// TIA Portal V16 program export: 1 tag tables, 0 data types, 0 data blocks, 2 code blocks (in call order from the OBs), 0 instance data blocks

VAR_GLOBAL   // PLC tag table "Default tag table"
END_VAR

ORGANIZATION_BLOCK "Main"   // OB1, LAD, ProgramCycle
TITLE = "Main Program Sweep (Cycle)"
{ S7_Optimized_Access := 'TRUE' }
VERSION : 0.1
// stored: AutoNumber true, IsIECCheckEnabled false, SetENOAutomatically false
BEGIN

REGION Network 1
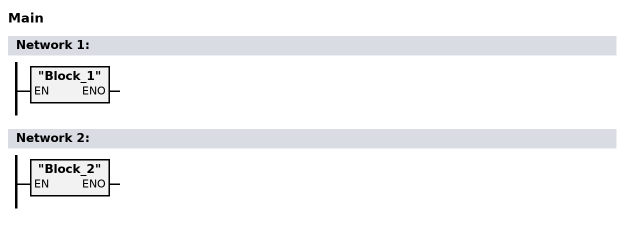
   RUNG wire#powerrail
      "Block_1"()
   END_RUNG
   // the same network as SCL:
   "Block_1"();
END_REGION

REGION Network 2
   RUNG wire#powerrail
      "Block_2"()
   END_RUNG
   // the same network as SCL:
   "Block_2"();
END_REGION
END_ORGANIZATION_BLOCK

FUNCTION "Block_1" : Void   // FC1, LAD
{ S7_Optimized_Access := 'TRUE' }
VERSION : 0.1
// stored: AutoNumber true, IsIECCheckEnabled false, SetENOAutomatically false, UDAEnableTagReadback false
BEGIN
END_FUNCTION
